# EPICS autosave request: iocBoot/ioc13idd/auto_settings_xps.req
file "CARS_motor_settings.req",         P=$(P), M=m81
file "CARS_motor_settings.req",         P=$(P), M=m82
file "CARS_motor_settings.req",         P=$(P), M=m83
file "CARS_motor_settings.req",         P=$(P), M=m84
